TYPE ST_ExampleDevice :
STRUCT
	//IO
	stAxis	:	AXIS_REF;
	i_xLoLim	AT %I*	:	BOOL;
	i_xHiLim	AT %I*	:	BOOL;
	
	//Supervisory System
	sc_eReqState	:	E_ExampleDeviceStates;
	sr_eState	:	E_ExampleDeviceStates;
END_STRUCT
END_TYPE

(* stored: Version 1.1.0.1, ProductVersion 3.1.4022.10
   DUT ST_ExampleDevice: Id {bc9ee667-91fb-46f2-af26-3ee8851b76e5} *)
